TYPE E_AlarmState :
(
	ActiveUnacknowledged			:= 1,
	InactiveUnacknowledged			:= 2,
	ActiveAcknowledged				:= 3,
	InactiveAcknowledged			:= 4
);
END_TYPE

(* stored: Version 1.1.0.1, ProductVersion 3.1.4024.9
   DUT E_AlarmState: Id {ba35f058-df8f-452b-9377-01da1bbe4bd7} *)
